INTERFACE ITask

METHOD Abort : BOOL
VAR_INPUT
END_VAR
END_METHOD

PROPERTY Busy : bool
GET
END_GET
END_PROPERTY

PROPERTY Done : bool
GET
END_GET
END_PROPERTY

PROPERTY Error : bool
GET
END_GET
END_PROPERTY

METHOD Execute : BOOL
VAR_INPUT
END_VAR
END_METHOD

END_INTERFACE

(* stored: Version 1.1.0.1, ProductVersion 3.1.4024.9
   Itf ITask: Id {fb28ad51-3810-4924-a43f-1a45d275c5a0}
   Method Abort: Id {009ea5f9-cf75-4404-a111-4f361e546ffe}
   Property Busy: Id {f9f7185f-c90d-4458-b002-32ecc21b7f06}
   Get Get: Id {55383a80-7455-4a83-9fec-915dce316c4d}
   Property Done: Id {8a73b454-d2ab-4126-8c8b-0a812fdd006c}
   Get Get: Id {23ec782b-9ddc-4d92-a2f4-de60da46c073}
   Property Error: Id {9cf6f3c6-739f-4607-866c-a636617ee49d}
   Get Get: Id {29dd3eb6-11d0-43dc-8804-c2ed97f85a7b}
   Method Execute: Id {2098d824-7923-42ba-b31d-914338060f7f} *)
